(* CoDeSys 2.3.9.62 project: SemaforoGRAFCET.pro *)
(* Libraries: Standard.lib 2.6.14 10:37:46, IecSfc.lib 2.6.14 10:37:46 *)

(* Global variable list: Global_Variables *)
VAR_GLOBAL

 (* Entradas *)
	M: BOOL;

      (*Salidas*)
	Rojo: BOOL;    	(* Luz roja*)
	Amarillo:BOOL;	(* Luz amarilla *)
	Verde:BOOL;		(* Luz verde *)
END_VAR

(* POU PLC_PRG, SFC *)
PROGRAM PLC_PRG
VAR
    (* declaración  de contadores *)
	CONTA: CTU;
END_VAR
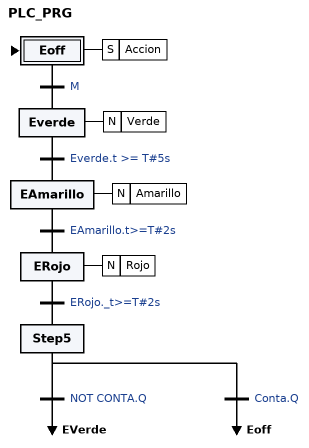
INITIAL_STEP Eoff:
	Accion(S);
END_STEP
TRANSITION FROM Eoff TO Everde := M;
END_TRANSITION
STEP Everde:
	Verde(N);
END_STEP
TRANSITION FROM Everde TO EAmarillo := Everde.t >= T#5s;
END_TRANSITION
STEP EAmarillo:
	Amarillo(N);
END_STEP
TRANSITION FROM EAmarillo TO ERojo := EAmarillo.t>=T#2s;
END_TRANSITION
STEP ERojo:
	Rojo(N);
END_STEP
TRANSITION FROM ERojo TO Step5 := ERojo._t>=T#2s;
END_TRANSITION
STEP Step5:
END_STEP
TRANSITION FROM Step5 TO EVerde := NOT CONTA.Q;
END_TRANSITION
TRANSITION FROM Step5 TO Eoff := Conta.Q;
END_TRANSITION
END_PROGRAM
ACTION Accion:
Conta(PV:=3, CU:=erojo.x, Reset:=Eoff.x);
END_ACTION

(* Visualisation SemaforoSimple
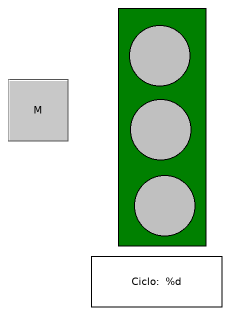
ellipse at (156,41)-(217,102): alarm colour if Rojo
ellipse at (157,115)-(218,176): alarm colour if Amarillo
ellipse at (161,191)-(222,252): alarm colour if Verde
rectangle at (118,272)-(249,323): text "Ciclo:  %d"; shows PLC_PRG.CONTA.CV
button at (35,95)-(95,157): text "M"; taps M
1 more shapes without text or variables
*)
